// TwinCAT 3 PLC project PLC01
// ProgramVersion: 3.1.4026.19
// CompilerDefines: VISU_USEPROPERTYINFO
// libraries:
//   Tc2_EtherCAT, * (Beckhoff Automation GmbH)
//   Tc2_Standard, * (Beckhoff Automation GmbH)
//   Tc2_System, * (Beckhoff Automation GmbH)
//   Tc2_Utilities, * (Beckhoff Automation GmbH)
// project tree:
//   DUTs/ st_SlaveInfo.TcDUT
//   / GlobalTextList.TcGTLO, PlcTask.TcTTO, Visualization Manager.TcVMO (not stored)
//   POUs/ MAIN.TcPOU, prgECatDiag.TcPOU
//   VISUs/ Visualization.TcVIS
// real-time tasks:
//   TASK PlcTask: cycle T#10ms, priority 20, ADS port 350
// I/O:
//   DEVICE Device 1 (EtherCAT), AmsNetId 10.199.162.27.2.1
//     Term 1 (EK1101) [EK1101 EtherCAT Coupler (2A E-Bus, ID switch)]
//       Term 2 (EL2008) [EL2008 8Ch. Dig. Output 24V, 0.5A]
//       Term 3 (EL2008) [EL2008 8Ch. Dig. Output 24V, 0.5A]
//       Term 4 (EL3702) [EL3702 2Ch. Ana. Input +/-10V, DIFF, Oversample]
//       Term 5 (EL9512) [EL9512 Power supply terminal 12V]
//       Term 6 (EL9011) [EL9011 End Terminal]
// variable links:
//   (this object) <-> Device 1 (EtherCAT)
//     PlcTask Inputs/prgECatDiag.netId <-> InfoData/AmsNetId
//   (this object) <-> Device 1 (EtherCAT)/Term 1 (EK1101)/Term 2 (EL2008)
//     PlcTask Outputs/prgECatDiag.bOut <-> Channel 1/Output

CONFIGURATION PLC01
    RESOURCE PLC ON TwinCAT3
        TASK PlcTask(INTERVAL := T#10ms, PRIORITY := 20);
        PROGRAM MAIN WITH PlcTask : MAIN;
    END_RESOURCE
END_CONFIGURATION

// ---- DUTs/st_SlaveInfo.TcDUT
TYPE st_SlaveInfo :
STRUCT
	configDevName, scannedDevName:STRING;
	addr:WORD;
	devState:STRING;
END_STRUCT
END_TYPE

// ---- POUs/MAIN.TcPOU
PROGRAM MAIN
VAR
END_VAR

prgECatDiag();

END_PROGRAM

// ---- POUs/prgECatDiag.TcPOU
PROGRAM prgECatDiag
VAR
	masterDiag: FB_EcGetMasterState;		//
	slaveState: FB_EcGetAllSlaveStates;     //
	getConfSlaves: FB_EcGetConfSlaves;      //
	getScannedSlaves: FB_EcGetScannedSlaves;//
	netId AT %I*:AMSNETID;
	bGetStates: BOOL;
	trigGetState: R_TRIG;
	iState: INT;
	sNetId: Tc2_EtherCAT.T_AmsNetId;
	state: WORD;
	nSlave: UINT;
	slavesBuffer: ARRAY[0..cMaxNumOfSlaves] OF ST_EcSlaveState;
	configuredSlaves: ARRAY [0..cMaxNumOfSlaves] OF ST_EcSlaveConfigData;
	nSlavesConf: UINT;
	nSlavesScanned: UINT;
	scannedSlaves: ARRAY [0..cMaxNumOfSlaves] OF ST_EcSlaveScannedData;
	asScannedProductNames: ARRAY[0..cMaxNumOfSlaves] OF STRING;
	i: UINT;
	bOut AT %Q*:BOOL;
	aSlaveInfo: ARRAY[0..cMaxNumOfSlaves] OF st_SlaveInfo;
END_VAR
VAR CONSTANT
	cMaxNumOfSlaves: UINT:=30;	//change as you which
	asEmptyStrings: ARRAY [0..cMaxNumOfSlaves] OF STRING;
END_VAR

trigGetState(CLK:=bGetStates);

IF trigGetState.Q THEN
	iState:=10;
	M_ResetSlaveNames();
END_IF
sNetId:= F_CreateAmsNetId(nIds:= netId);
CASE iState OF
	0:
		;
	10:
		masterDiag(
			sNetId:= sNetId, 
			bExecute:= TRUE, 
			tTimeout:=T#3S , 
			state=> state);
		IF NOT masterDiag.bBusy AND NOT masterDiag.bError THEN
			iState:=20;
		END_IF
	20:
		slaveState(
			sNetId:= sNetId, 
			pStateBuf:= ADR(slavesBuffer), 
			cbBufLen:= SIZEOF(slavesBuffer), 
			bExecute:= TRUE,
			nSlaves=>nSlave );
		IF NOT slaveState.bBusy AND NOT slaveState.bError THEN
			iState:=30;
		END_IF
	30:
		getConfSlaves(
			sNetId:= sNetId, 
			pArrEcConfSlaveInfo:=ADR(configuredSlaves) , 
			cbBufLen:= SIZEOF(configuredSlaves), 
			bExecute:= TRUE, 
			nSlaves=> nSlavesConf);
		IF NOT getConfSlaves.bBusy AND NOT getConfSlaves.bError THEN
			iState:=40;
		END_IF
	40:
		getScannedSlaves(
			bExecute:=TRUE , 
			sNetId:= sNetId, 
			pArrEcScannedSlaveInfo:=ADR(scannedSlaves) , 
			cbBufLen:=SIZEOF(scannedSlaves) , 
			nSlaves=>nSlavesScanned );
		IF NOT getScannedSlaves.bBusy AND NOT getScannedSlaves.bError THEN
			iState:=50;
			FOR i:= 0 TO cMaxNumOfSlaves DO
				IF scannedSlaves[i].stSlaveIdentity.productCode <> 0 THEN
					//asScannedProductNames[i]:= ;
					aSlaveInfo[i].configDevName:=configuredSlaves[i].sName;
					aSlaveInfo[i].addr:=configuredSlaves[i].nAddr;
					aSlaveInfo[i].scannedDevName:= F_ConvProductCodeToString(scannedSlaves[i].stSlaveIdentity);
					aSlaveInfo[i].devState:= F_ConvSlaveStateToString(slavesBuffer[i]);
				ELSE
					EXIT;
				END_IF
			END_FOR
		END_IF
	50:
		iState:=0;
END_CASE
bOut:=TRUE;

METHOD M_ResetSlaveNames
VAR_INPUT
END_VAR
memcpy(ADR(asScannedProductNames), ADR(asEmptyStrings),SIZEOF(asEmptyStrings));
END_METHOD

END_PROGRAM

// ---- GlobalTextList.TcGTLO
TEXTLIST GlobalTextList
  551 = 'Endereço'
  209 = 'Estado'
  525 = 'Link'
  963 = 'Link Status'
  486 = 'Name'
  851 = 'Nome'
  733 = 'Nome escaneado'
  203 = 'ReadSlaves'
  812 = 'Tipo'
END_TEXTLIST

// ---- VISUs/Visualization.TcVIS
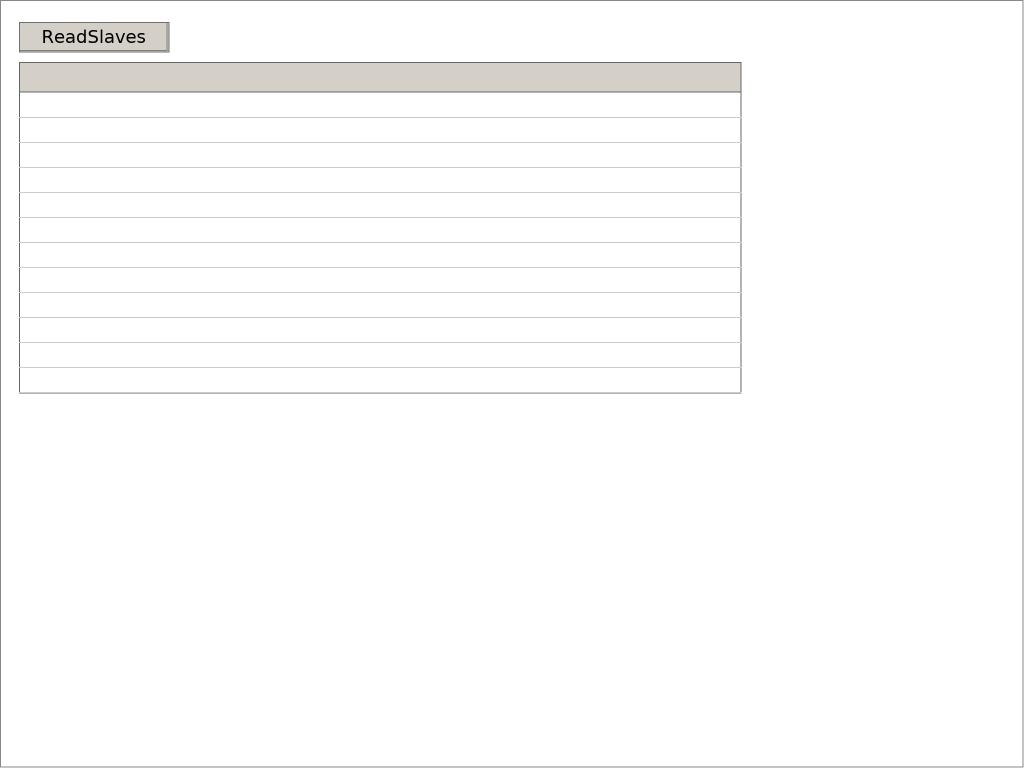
VISUALIZATION Visualization  // 1024x768
    Button (19,22 150x30), "ReadSlaves"
        tap prgECatDiag.bGetStates
    Table (19,62 722x331), data array: prgECatDiag.aSlaveInfo
        p1014161805: PRGECATDIAG.cMaxNumOfSlaves - 0 + INT#1
        p3854506369: prgECatDiag.aSlaveInfo[INDEX].configDevName
        p1892666644: prgECatDiag.aSlaveInfo[INDEX].scannedDevName
        p338671338: prgECatDiag.aSlaveInfo[INDEX].addr
        p2170511999: prgECatDiag.aSlaveInfo[INDEX].devState
        p511219082: Nome escaneado
        p1755163831: Endereço
        p4092479075: Estado
END_VISUALIZATION
